(* PLC project PowerFlex525_in_progress.project, CODESYS CODESYS V3.5 SP22 Patch 2 *)
(* stored: creationDateTime 2026-07-29T18:04:08.9142058, modificationDateTime 2026-07-29T17:57:32.3508621 *)

PROGRAM PLC_PRG
  VAR
    fbModuleBinding : TF_Codesys_ENIP_ModuleBinding;
    fbReconfigure : DED.Reconfigure;
    xInp_Inhibit : BOOL;
    xInp_Uninhibit : BOOL;
    xInp_Connected : BOOL;
    xInp_Enabled : BOOL;
    xInp_Faulted : BOOL;
    xInp_DiagnosticAvailable : BOOL;
    xInp_CanReconfigure : BOOL;
    xInp_ReconfigureBusy : BOOL;
    xInp_ReconfigureDone : BOOL;
    xInp_ReconfigureFailed : BOOL;
    xOut_Connected : BOOL;
    xOut_Enabled : BOOL;
    xOut_Faulted : BOOL;
    xOut_DiagnosticAvailable : BOOL;
    xOut_RequestReconfigure : BOOL;
    xOut_RequestedEnable : BOOL;
    xOut_ReconfigureBlocked : BOOL;
    xOut_ReconfigureBusy : BOOL;
    xOut_ReconfigureDone : BOOL;
    xOut_ReconfigureFailed : BOOL;
    xObservedEnabled : BOOL;
    xObservedDiagnosticAvailable : BOOL;
    sObservedDiagnostic : STRING(255);
    eObservedDeviceState : DED.DEVICE_STATE;
    eObservedReconfigureError : DED.ERROR;
  END_VAR

                  xObservedEnabled := Dev_PF525.Enable;
xObservedDiagnosticAvailable := Dev_PF525.xDiagnosticAvailable;
sObservedDiagnostic := Dev_PF525.sDiagString;
eObservedDeviceState := Dev_PF525.GetDeviceState();

xInp_CanReconfigure :=
    DED.CanReconfigure(itfNode := Dev_PF525);
    
xInp_Connected :=
    (Dev_PF525.eState = IoDrvEtherNetIP.AdapterState.RUNNING)
    AND
    (eObservedDeviceState = DED.DEVICE_STATE.RUNNING);

xInp_Enabled := Dev_PF525.Enable;

xInp_Faulted :=
    (Dev_PF525.eState = IoDrvEtherNetIP.AdapterState.BUS_ERROR)
    OR
	(Dev_PF525.eState = IoDrvEtherNetIP.AdapterState.ERROR)
    OR
    (eObservedDeviceState = DED.DEVICE_STATE.ERROR);

xInp_DiagnosticAvailable :=
    Dev_PF525.xDiagnosticAvailable;
	
xInp_ReconfigureBusy :=
    fbReconfigure.xBusy;

xInp_ReconfigureDone :=
    fbReconfigure.xDone;

xInp_ReconfigureFailed :=
    fbReconfigure.xError;

eObservedReconfigureError :=
    fbReconfigure.eError;

fbModuleBinding(
    Inp_Connected := xInp_Connected,
    Inp_Enabled := xInp_Enabled,
    Inp_Faulted := xInp_Faulted,
    Inp_DiagnosticAvailable := xInp_DiagnosticAvailable,
    Inp_CanReconfigure := xInp_CanReconfigure,
    Inp_ReconfigureBusy := xInp_ReconfigureBusy,
    Inp_ReconfigureDone := xInp_ReconfigureDone,
    Inp_ReconfigureFailed := xInp_ReconfigureFailed,
    Inp_Inhibit := xInp_Inhibit,
    Inp_Uninhibit := xInp_Uninhibit,
    Out_Connected => xOut_Connected,
    Out_Enabled => xOut_Enabled,
    Out_Faulted => xOut_Faulted,
    Out_DiagnosticAvailable => xOut_DiagnosticAvailable,
    Out_RequestReconfigure => xOut_RequestReconfigure,
    Out_RequestedEnable => xOut_RequestedEnable,
    Out_ReconfigureBlocked => xOut_ReconfigureBlocked,
    Out_ReconfigureBusy => xOut_ReconfigureBusy,
    Out_ReconfigureDone => xOut_ReconfigureDone,
    Out_ReconfigureFailed => xOut_ReconfigureFailed
);

IF xOut_RequestReconfigure THEN
    Dev_PF525.Enable := xOut_RequestedEnable;
END_IF;

fbReconfigure(
    xExecute := xOut_RequestReconfigure,
    itfNode := Dev_PF525
);


                
END_PROGRAM

FUNCTION_BLOCK TF_Codesys_ENIP_ModuleBinding
  VAR_INPUT
    Inp_Connected : BOOL;
    Inp_Enabled : BOOL;
    Inp_Faulted : BOOL;
    Inp_DiagnosticAvailable : BOOL;
    Inp_CanReconfigure : BOOL;
    Inp_ReconfigureBusy : BOOL;
    Inp_ReconfigureDone : BOOL;
    Inp_ReconfigureFailed : BOOL;
    Inp_Inhibit : BOOL;
    Inp_Uninhibit : BOOL;
  END_VAR
  VAR_OUTPUT
    Out_Connected : BOOL;
    Out_Enabled : BOOL;
    Out_Faulted : BOOL;
    Out_DiagnosticAvailable : BOOL;
    Out_RequestReconfigure : BOOL;
    Out_RequestedEnable : BOOL;
    Out_ReconfigureBlocked : BOOL;
    Out_ReconfigureBusy : BOOL;
    Out_ReconfigureDone : BOOL;
    Out_ReconfigureFailed : BOOL;
  END_VAR
  VAR
    CommandLatch : BOOL;
  END_VAR

                  Out_Connected := Inp_Connected;
Out_Enabled := Inp_Enabled;
Out_Faulted := Inp_Faulted;
Out_DiagnosticAvailable := Inp_DiagnosticAvailable;
Out_ReconfigureBusy := Inp_ReconfigureBusy;
Out_ReconfigureDone := Inp_ReconfigureDone;
Out_ReconfigureFailed := Inp_ReconfigureFailed;
Out_RequestReconfigure := FALSE;
IF ((Inp_Inhibit OR Inp_Uninhibit) AND NOT (CommandLatch)) THEN
    IF (Inp_CanReconfigure AND NOT (Inp_ReconfigureBusy)) THEN
        Out_RequestedEnable := NOT (Inp_Inhibit);
        Out_RequestReconfigure := TRUE;
        Out_ReconfigureBlocked := FALSE;
    ELSE
        Out_ReconfigureBlocked := TRUE;
    END_IF;
END_IF;
IF Inp_ReconfigureDone THEN
    Out_ReconfigureBlocked := FALSE;
END_IF;
CommandLatch := (Inp_Inhibit OR Inp_Uninhibit);
                
END_FUNCTION_BLOCK

CONFIGURATION Application
  RESOURCE Application ON PLC
    TASK MainTask(INTERVAL := T#20ms, PRIORITY := 1);
    PROGRAM PLC_PRG WITH MainTask : PLC_PRG;
  END_RESOURCE
END_CONFIGURATION
